// TIA Portal V20 export
TYPE "UDT_ConfigPaletizador"
   STRUCT
      VeloManual : Int := 1000;   // Velocidad en Manual
      VeloCapa : Int := 2000;   // Velocidad de Movimiento de Capa
      VeloRapidaDown : Int := 5000;   // Velocidad Rapida de Movimiento Down
      VeloLentaDown : Int := 3000;   // Velocidad Lenta de Movimiento Down
      VeloRapidaUp : Int := 8000;   // Velocidad Rapida de Movimiento Up
      VeloLentaUp : Int := 2000;   // Velocidad Lenta de Movimiento Up
      PosVeloLentaDown : Int := 500;   // Posicion al final para entrada en Lenta en MOv. Down
      PosVeloLentaUp : Int := 500;   // Posicion al final para entrada en Lenta en MOv. Up
      AlturaMax : Int := 3490;   // Altura MAx de Posicion del elevador
      AlturaMin : Int := 300;   // Altura Min de Posicion del Elevador
      AlturaPaleta : Int := 140;   // Altura de Paleta
      AlturaGalibo : Int := 2370;   // Altura de Control de Mov al Puesto
      AlturaBarrera : Int := 3900;   // Altura de la Paleta en el Nivel (Dinamico)
      PosicionCarga : Int := 350;   // Altura de Carga de Paleta
      PosicionDesCarga : Int := 350;   // Altura de DesCarga de Paleta
      AlturaPedido : Int := 1200;
   END_STRUCT;
END_TYPE
